(*
Casts I_Component to I_Arg
*)
FUNCTION ICompToIArg : Result
VAR_INPUT
	iSource	: I_Component;
END_VAR
VAR_OUTPUT
	iDest	: I_Arg;
END_VAR

IF iSource = 0 THEN
	ICompToIArg := Err.Itf0;
	RETURN;
END_IF

IF __QUERYINTERFACE(iSource, iDest) THEN
	ICompToIArg := Ok;
ELSE
	iDest := 0;
	ICompToIArg := Err.NoMatch;
END_IF

END_FUNCTION

(* stored: Version 1.1.0.1
   POU ICompToIArg: Id {cea0c7a0-5752-446d-bb01-5581ac3b101a}, SpecialFunc None *)
